FUNCTION fc_Set_DT : DT
VAR_INPUT
	year 	: INT;
	month 	: INT;
	day 	: INT;
	hour 	: INT;
	minute 	: INT;
	second 	: INT;
END_VAR
VAR
END_VAR

fc_Set_DT := DWORD_TO_DT(DATE_TO_DWORD(fc_Set_Date(YEAR, MONTH, day)) + INT_TO_DWORD(SECOND) + INT_TO_DWORD(MINUTE) * 60 + INT_TO_DWORD(HOUR) * 3600);

END_FUNCTION

(* stored: Version 1.1.0.1, ProductVersion 3.1.4024.11
   POU fc_Set_DT: Id {e2b77e93-efdf-4572-9bc0-5191c4c05af5}, SpecialFunc None *)
